{attribute 'strict'}
TYPE E_CognexCameraResetSystemStatus :
(
	WAITING_FOR_STATUS_CODE					:= 2,	
	THE_COMMAND_WAS_EXECUTED_SUCCESSFULLY	:= -1,
	USER_DOES_NOT_HAVE_FULL_ACCESS			:= -6
);
END_TYPE

(* stored: Version 1.1.0.1, ProductVersion 3.1.4024.9
   DUT E_CognexCameraResetSystemStatus: Id {4068e00c-9278-4a9e-8f7c-d0cca12c1b7b} *)
